PROGRAM prg_jafunctie
VAR
	Ingang		AT		%I*		:BOOL;
	Uitgang		AT		%Q*		:BOOL;
END_VAR

Uitgang := Ingang;

END_PROGRAM

(* stored: Version 1.1.0.1, ProductVersion 3.1.4024.15
   POU prg_jafunctie: Id {672652f4-dbb3-4fa0-8d2f-9da87f6e4f8c}, SpecialFunc None *)
